// ---- VISUs/Visualization.TcVIS
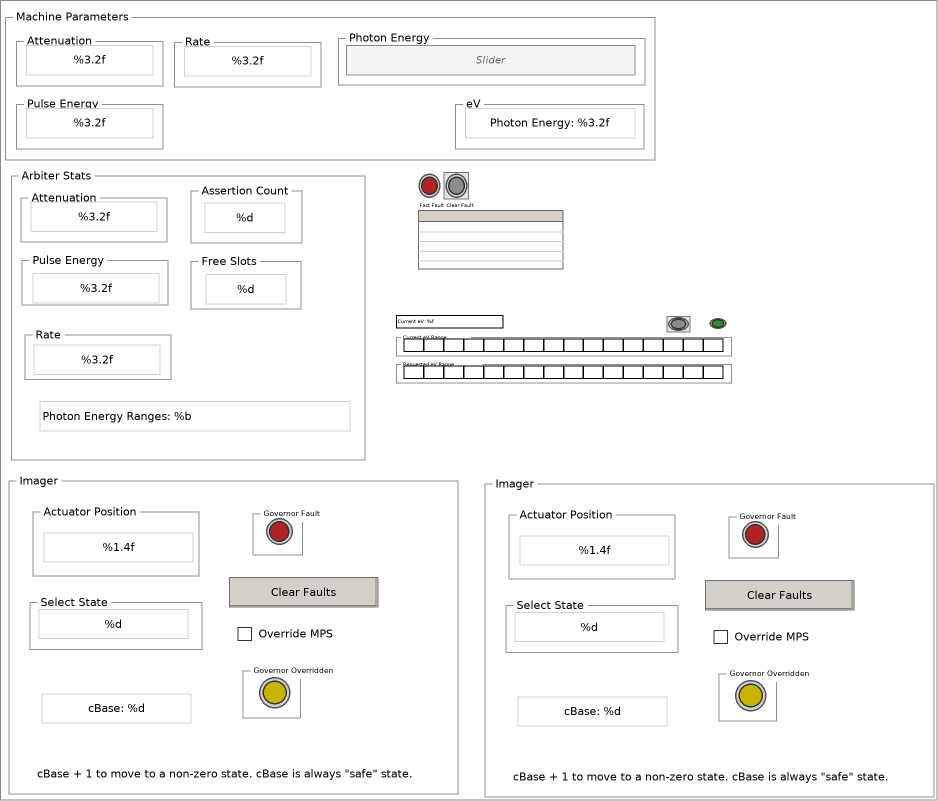
VISUALIZATION Visualization  // 938x801
    GroupBox (5,9 650x151), "Machine Parameters"
        GroupBox (11,24 147x53), "Attenuation"
            Textfield (10,12 127x30), "%3.2f", text variable: PMPS_GVL_BeamParams.stCurrentBeamParameters.fAtt
        GroupBox (11,87 147x53), "Pulse Energy"
            Textfield (10,12 127x30), "%3.2f", text variable: PMPS_GVL_BeamParams.stCurrentBeamParameters.fPP_mJ
        GroupBox (169,25 147x53), "Rate"
            Textfield (10,12 127x30), "%3.2f", text variable: PMPS_GVL_BeamParams.stCurrentBeamParameters.nRate
        GroupBox (333,21 307x55), "Photon Energy"
            Slider (8,15 289x30), variable: MachineSimulation.fbMachine.i_reV, scale 0..1600
        GroupBox (450,87 189x53), "eV"
            Textfield (10,12 170x30), "Photon Energy: %3.2f", text variable: PMPS_GVL_BeamParams.stCurrentBeamParameters.reV
    Frame (6,468 454x328)
        shows ImagerGUI(fbDevice := MAIN.fbDev1)
    Frame (482,471 454x328)
        shows ImagerGUI(fbDevice := MAIN.fbDev2)
    Frame (417,172 147x98)
        shows FastFaultGUI(FastFault := GVL.g_FastFaultOutput1)
    Frame (11,168 356x294)
        shows ArbiterStats(fbArbiter := GVL.g_fbArbiter)
    Frame (396,315 337x69)
        shows PhotonEnergyWatcher(Watcher := PMPS_Arbiter.fbPhotonEnergyWatcher)
END_VISUALIZATION

// ---- VISUs/WordBitDisplay.TcVIS
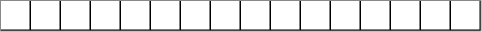
VISUALIZATION WordBitDisplay  // 482x32
VAR_IN_OUT
	nVal	:	WORD;
END_VAR
    Rectangle (0,0 30x30), colour toggle: nVal.15
    Rectangle (30,0 30x30), colour toggle: nVal.14
    Rectangle (60,0 30x30), colour toggle: nVal.13
    Rectangle (90,0 30x30), colour toggle: nVal.12
    Rectangle (120,0 30x30), colour toggle: nVal.11
    Rectangle (150,0 30x30), colour toggle: nVal.10
    Rectangle (180,0 30x30), colour toggle: nVal.9
    Rectangle (210,0 30x30), colour toggle: nVal.8
    Rectangle (240,0 30x30), colour toggle: nVal.7
    Rectangle (270,0 30x30), colour toggle: nVal.6
    Rectangle (300,0 30x30), colour toggle: nVal.5
    Rectangle (330,0 30x30), colour toggle: nVal.4
    Rectangle (360,0 30x30), colour toggle: nVal.3
    Rectangle (390,0 30x30), colour toggle: nVal.2
    Rectangle (420,0 30x30), colour toggle: nVal.1
    Rectangle (450,0 30x30), colour toggle: nVal.0
END_VISUALIZATION
